{attribute 'Tc2GVLVarNames'}
VAR_GLOBAL
	bstart					:BOOL;
	bSet					:BOOL;
	bstop                   :BOOL;
	
	RealLaserD				AT %I*	 :UINT;
	RealVelocimeterD      	AT %I*   :UINT;
	EncoderD           			   :LREAL;
	
	
	laserSetPoint					:UINT;
	LaserD							:UINT;
	
	VelocimeterSetPoint				:UINT;
	VelocimeterD                    :UINT;
	
	
	Reel					:AXIS_REF;
	
	
	bSetBTN			AT %I*	   	:BOOL;
	bStartBTN       at %I*       :bool;
	bStopBTN        at %I*       :bool;
END_VAR

(* stored: Version 1.1.0.1, ProductVersion 3.1.4024.12
   GVL Standard: Id {83f8f447-0eb1-4d0c-b486-f84fc99139ff} *)
